(* IEC 61131-3 sources: UniTest/UniTest_br/Library_tests/test_assertLessEqual_DWORD, 2 files *)

(* ---- LocalVariables.var ---- *)
VAR
    vTestCases : ARRAY[0..20] OF utTestCase; (*Definition of all test cases for this POU*)
    testRunner : utTestSuite; (*Test Suite fb instance to run the tests*)
    vRunAll : BOOL; (*Manual command to run all tests for this POU*)
    vResetAll : BOOL; (*Manual command to reset all tests for this POU*)
    vTestCase1_act : DWORD; (*Test data 1 of test case 1*)
    vTestCase1_xp : DWORD; (*Test data 2 of test case 1*)
    vTestCase2_act : DWORD; (*Test data 1 of test case 2*)
    vTestCase2_xp : DWORD; (*Test data 2 of test case 2*)
    vTestCase3_act : DWORD; (*Test data 1 of test case 3*)
    vTestCase3_xp : DWORD; (*Test data 2 of test case 3*)
END_VAR

(* ---- main.st ---- *)
PROGRAM _CYCLIC
    (*https://github.com/tkucic/UniTest/blob/main/docs/docs/ns/Library_tests/prg/test_assertLessEqual_DWORD.md*)
    (*Run the test cases*)
    TEST_CASE_1_SETUP;
    TEST_CASE_1_EXEC;

    TEST_CASE_2_SETUP;
    TEST_CASE_2_EXEC;

    TEST_CASE_3_SETUP;
    TEST_CASE_3_EXEC;

    (*Instantiate the test runner*)
    testRunner(
    	Id := 118,
    	Name := 'assertLessEqual_DWORD',
        RunTests := gRunAll OR vRunAll,
    	ResetTests := gResetAll OR vResetAll,
    	TestCases:=vTestCases);

    (*Report the results to the collection global*)
    gResults[testRunner.Id] := testRunner.Summary;
END_PROGRAM
